PROGRAM VARINFO

VAR
    MyVarInfo : __SYSTEM.VAR_INFO;
    nVar      : INT;
END_VAR

MyVarInfo := __VARINFO(nVar);

END_PROGRAM

(* stored: Version 1.1.0.1, ProductVersion 3.1.4024.12
   POU VARINFO: Id {dccb941f-2b41-458b-a0fe-fa3962edb20e}, SpecialFunc None *)
